// TIA Portal V16 export
// export: Created 2022-12-12T13:38:05.5321597Z, ExportSetting WithDefaults, DisplayName Totally Integrated Automation Portal, DisplayVersion V16 Update 6, DisplayName TIA Portal Version Control Interface, DisplayVersion V16 Update 2, DisplayName TIA Portal Openness, DisplayVersion V16 Update 6, DisplayName SINAMICS Startdrive Advanced, DisplayVersion V16 Update 5, DisplayName SINAMICS Startdrive G130, G150, S120, S150, SINAMICS MV, S210, DisplayVersion V16 Update 5, DisplayName SINAMICS Startdrive G110M, G120, G120C, G120D, G120P, G115D, DisplayVersion V16 Update 5, DisplayName STEP 7 Professional, DisplayVersion V16 Update 6, DisplayName STEP 7 Safety, DisplayVersion V16, DisplayName WinCC Advanced, DisplayVersion V16 Update 6
DATA_BLOCK "Centrador_Paletes_DB"   // DB11
VERSION : 0.1
// stored: AutoNumber true, InstanceOfName Centrador_Paletes, InstanceOfType FB
"Centrador_Paletes"
   // VAR_INPUT
   //    Centrador_Aberto_1 : Bool;
   //    Centrador_Aberto_2 : Bool;
   //    Detetor_Palete : Bool;
   //    Palete_Centrada_1 : Bool;
   //    Palete_Centrada_2 : Bool;
   // END_VAR
   // VAR_OUTPUT
   //    "ETAPA 1 (INICIO)" : Bool;
   //    "ETAPA 2" : Bool;
   //    "ETAPA 3" : Bool;
   //    "ETAPA 4" : Bool;
   //    Motor_Tapete_Centrador : Bool;
   //    Motor_Centrador_Sentido_Direto : Bool;
   //    Motor_Centrador_Sentido_Inverso : Bool;
   // END_VAR
BEGIN
END_DATA_BLOCK
